INTERFACE I_RegisterMover

METHOD RegisterMover : BOOL
VAR_INPUT
	mover : I_Mover;
END_VAR
END_METHOD

END_INTERFACE

(* stored: Version 1.1.0.1
   Itf I_RegisterMover: Id {4b37523f-2df6-41ad-92b4-6134a7e08087}
   Method RegisterMover: Id {456afb0d-cc9d-417a-b09b-6924221316a8} *)
